FUNCTION_BLOCK FB_FaultHandler
(* 
The faulthandler is responsible for 
	- providing the means for objects to register their faults
	- reporting the active fault types (i.e., message, fatal fault, etc.) --> arActiveFaultTypes
	- providing the means to reset a fault type
	- keeping a log of all faults

It is not responsible for
	- resetting the actual fault (this is up to the object that registered the fault)
	- handling any HMI related functionality

Active faults do not disappear from the log, the need to be manually cleared by issuing a CmdReset and CmdClearInactive.
*)
VAR CONSTANT
	MAX_FAULTS_IN_LOG : UINT := 10;
END_VAR
VAR_INPUT
	nMaxInactiveCycles : UINT := 50; // Once faults haven't been activated for a number of PLC cycles, deactivate them. 0 = do not automatically deactivate faults 
END_VAR
VAR_OUTPUT
	arFaultLog 			: ARRAY [1..MAX_FAULTS_IN_LOG] OF UDT_FaultLogItem;
	nFaultsInLog 		: UINT;
	nActiveFaults 		: UINT;
	arActiveFaultTypes 	: ARRAY[0..(E_FaultTypes._ENUM_SIZE - 1)] OF BOOL; // Status of each fault type
END_VAR
VAR
	bCmdReset : BOOL;
	eResetState : E_ResetState;
	arActiveFaultTypes_Internal : ARRAY[0..(E_FaultTypes._ENUM_SIZE - 1)] OF BOOL; // The actual status of each fault type, which is reported unless the reset cycle is active
	
	nLogIndex : UINT; // Array index of the last added item in the log (zero until the first item arrives)
	nIterIndex : UINT; // Index of the fault log iterator (used for properties First and Next)
END_VAR

UpdateInactiveCycles();

ExecReset();

UpdateActiveFaultStatus();

METHOD PUBLIC CmdAddFault : BOOL
(*
CmdAddFault should be called every cycle.
If the fault is active, it's corresponding fault type is enabled.
Updates the fault log.
*)
VAR_IN_OUT
	stFault : UDT_Fault; // active fault structure input
END_VAR
VAR_INPUT
	stIdentity : UDT_Identity;
END_VAR
// Update the log
UpdateLog(stFault, stIdentity);
END_METHOD

METHOD PUBLIC CmdClearInactive : BOOL // Remove inactive faults from the log
VAR
	stEmptyItem : UDT_FaultLogItem;
	i : UINT; // Iterator
END_VAR
nFaultsInLog := MAX_FAULTS_IN_LOG;
IF (eResetState = E_ResetState.Idle) THEN
	FOR i := 1 TO MAX_FAULTS_IN_LOG DO
		IF (NOT arFaultLog[i].stFault.Active) THEN
			nFaultsInLog :=nFaultsInLog - 1;
			arFaultLog[i] := stEmptyItem;
			arFaultLog[i].bEmpty := TRUE;
		END_IF
	END_FOR
	CmdClearInactive := TRUE;
ELSE
	CmdClearInactive := FALSE;
END_IF
END_METHOD

METHOD PUBLIC CmdReset : BOOL // Reset faults; caller is responsible for stopping the call once TRUE is returned
VAR_INPUT
END_VAR
// Trigger the reset cycle
IF (eResetState = E_ResetState.Idle) THEN
	bCmdReset := TRUE;
END_IF

CmdReset := (eResetState = E_ResetState.Done); // Let the caller know when the reset cycle is finished
END_METHOD

METHOD PRIVATE ExecReset : BOOL
VAR
	i : UINT; // Iterator
END_VAR
CASE eResetState OF
	E_ResetState.Idle: // Wait for reset command
		IF bCmdReset THEN
			// Start the reset cycle
			bCmdReset := FALSE;
			eResetState := E_ResetState.ResetFaultTypes;
		ELSE
			ReportActiveFaultStatus();
		END_IF
	E_ResetState.ResetFaultTypes: 
		// During a reset, the active fault types are not updated 
		// This avoids that faults are not reported for 1 PLC cycle, even though they are still active
		// We do however clear the internal fault types, which are updated automatically during the WaitForFaults state.
		FOR i:= 0 TO (E_FaultTypes._ENUM_SIZE - 1) DO		
			arActiveFaultTypes_Internal[i] := FALSE;
		END_FOR
		eResetState := E_ResetState.WaitForFaults;

	E_ResetState.WaitForFaults: // Allow the PLC one cycle to re-add faults
		eResetState := E_ResetState.Done;

	E_ResetState.Done: // Done, report & allow caller one cycle to reset itself
		ReportActiveFaultStatus();
		eResetState := E_ResetState.Idle;
END_CASE
END_METHOD

METHOD PRIVATE FindNonEmptyFault : UINT // Update nIterIndex to first non-empy fault (if available)
VAR_INPUT
	nStartIndex : UINT;
END_VAR
VAR
	i : UINT; // Iterator
END_VAR
// Sanitize input
nStartIndex := LIMIT(1, nStartIndex, MAX_FAULTS_IN_LOG);

// Iterate array backwards until a non empty item is found.
FOR i := 1 TO MAX_FAULTS_IN_LOG DO
	IF arFaultLog[nStartIndex].bEmpty THEN
		nStartIndex := nStartIndex - 1;
		IF nStartIndex = 0 THEN
			nStartIndex := MAX_FAULTS_IN_LOG;
		END_IF
	ELSE
		EXIT;
	END_IF
END_FOR

FindNonEmptyFault := nStartIndex;
END_METHOD

PROPERTY PUBLIC Head : UDT_FaultLogItem // Returns the head of the log (the latest item added)
GET
nIterIndex := FindNonEmptyFault(nLogIndex);
Head := arFaultLog[nIterIndex];
END_GET
SET
END_SET
END_PROPERTY

PROPERTY PUBLIC Next : UDT_FaultLogItem // Get the next item in the log (travelling backwards through the array)
GET
nIterIndex := FindNonEmptyFault(nIterIndex - 1);
Next := arFaultLog[nIterIndex];
END_GET
SET
END_SET
END_PROPERTY

METHOD PRIVATE ReportActiveFaultStatus : BOOL // Update active fault types based on active faults in the log
VAR
	i : UINT; // Iterator
END_VAR
// Report the status of each fault type to outside world	
FOR i:= 0 TO (E_FaultTypes._ENUM_SIZE - 1) DO		
	arActiveFaultTypes[i] := arActiveFaultTypes_Internal[i];
END_FOR
END_METHOD

METHOD PRIVATE UpdateActiveFaultStatus : BOOL // Update active fault types based on active faults in the log
VAR
	i : UINT; // Iterator
END_VAR
// Get active faults from log
nActiveFaults := 0;
FOR i := 1 TO MAX_FAULTS_IN_LOG DO
	IF (arFaultLog[i].stFault.Active) THEN 
		// Update the number of active faults
		nActiveFaults := nActiveFaults + 1;
		// Update active fault type feedback
		arActiveFaultTypes_Internal[arFaultLog[i].stFault.FaultType] := TRUE; 
	END_IF
END_FOR
END_METHOD

METHOD PRIVATE UpdateInactiveCycles : BOOL // Update the number of inactive cycles, and deactive fault once it reaches the max number of inactive cycles
VAR
	i : UINT; // Iterator
END_VAR
IF (nMaxInactiveCycles > 0) THEN
	FOR i := 1 TO MAX_FAULTS_IN_LOG DO
		IF arFaultLog[i].stFault.Active THEN
			arFaultLog[i].nInactiveCycles := MIN(16#FFFF, arFaultLog[i].nInactiveCycles + 1);
			IF (arFaultLog[i].nInactiveCycles > nMaxInactiveCycles) THEN
				arFaultLog[i].stFault.Active := FALSE;
				arFaultLog[i].EndTime := Sys_Variables.SystemTime;	
			END_IF
		END_IF
	END_FOR
END_IF
END_METHOD

METHOD PRIVATE UpdateLog : BOOL
(*
Update the fault log array. 
If a fault becomes active, it is added to the array and the start time is updated.
If a fault stops being active, the end time is updated.
Inactive faults are cleared by CmdReset.
*)
VAR_IN_OUT
	stFault : UDT_Fault;
END_VAR
VAR_INPUT
	stIdentity : UDT_Identity;
END_VAR
VAR
	sId : STRING;
	nFaultIndexInLog : UINT;
	i : UINT; // Iterator
END_VAR
// Check if the fault already exists in the log. 
// For this, we need to compare the description and the fault ID.

// First, build the fault ID
sId := TO_STRING(stFault.FaultType);
sId := CONCAT(sId,'.');
IF stIdentity.nParentId > 0 THEN
	sId := CONCAT(sId,UDINT_TO_STRING(stIdentity.nParentId));
	sId := CONCAT(sId,'.');
END_IF
sId := CONCAT(sId,UINT_TO_STRING(stIdentity.nId));
sId := CONCAT(sId,'.');
sId := CONCAT(sId,UDINT_TO_STRING(stIdentity.eComponentType));
sId := CONCAT(sId,'.');
sId := CONCAT(sId,stIdentity.sName);

// Now check if the fault already exists in the log
FOR i := 1 TO MAX_FAULTS_IN_LOG DO
	IF (NOT arFaultLog[i].bEmpty) 
		AND (arFaultLog[i].Id = sId) 
		AND (arFaultLog[i].stFault.Description = stFault.Description)
		AND (ANY_TO_DWORD(arFaultLog[i].EndTime) = 0)
	THEN // Found fault in the log
		nFaultIndexInLog := i;
		EXIT; // No need to iterate any further
	END_IF
END_FOR

IF nFaultIndexInLog > 0 THEN // Already exists in the log
	IF (stFault.Active) THEN // Still active, reset inactive cycle counter
		arFaultLog[nFaultIndexInLog].nInactiveCycles := 0;
	ELSIF (ANY_TO_DWORD(arFaultLog[nFaultIndexInLog].EndTime) = 0) THEN // No longer active, update end time and active state
		arFaultLog[nFaultIndexInLog].stFault.Active := FALSE;
		arFaultLog[nFaultIndexInLog].EndTime := Sys_Variables.SystemTime;
	END_IF
ELSIF stFault.Active THEN // New active fault, add it to the log
	// Update the log index (if full, move to beginning of the log)
	nLogIndex := (nLogIndex MOD MAX_FAULTS_IN_LOG) + 1;
	nFaultsInLog := MIN(nFaultsInLog + 1, MAX_FAULTS_IN_LOG);
	// Copy to log and update start time
	arFaultLog[nLogIndex].bEmpty := FALSE;
	arFaultLog[nLogIndex].stFault := stFault;
	arFaultLog[nLogIndex].Id := sId;
	arFaultLog[nLogIndex].StartTime := Sys_Variables.SystemTime;
	arFaultLog[nLogIndex].EndTime := ANY_TO_DT(0);
	arFaultLog[nLogIndex].nInactiveCycles := 0;
END_IF
END_METHOD

END_FUNCTION_BLOCK

(* stored: Version 1.1.0.1, ProductVersion 3.1.4024.11
   POU FB_FaultHandler: Id {08f65884-c647-4a29-b7ba-51d088979c07}, SpecialFunc None
   Folder Private: Id {2e728eb6-79bc-4de8-8875-9d08a8df9edd}
   Method CmdAddFault: Id {cd103280-aca4-4b4a-a070-10b84eec5ffb}
   Method CmdClearInactive: Id {3ab26ba4-92e5-0c92-3fbe-58c7f26971b2}
   Method CmdReset: Id {a9c5d6bc-61dd-41fc-99d9-5b14d5fa2712}
   Method ExecReset: Id {5409ab96-3bb3-0061-05e8-ad57d1261a31}
   Method FindNonEmptyFault: Id {f653cfda-c6a2-0aba-0999-a219be313e66}
   Property Head: Id {51df95bf-2d5c-0e2f-1669-066486ace38d}
   Get Get: Id {5da39590-30a9-04b4-307b-1dd3ceac2537}
   Set Set: Id {f26a9a04-102d-0fab-2b21-bb756981a144}
   Property Next: Id {3bc770ea-8ea7-000b-0986-7649ccc14e3e}
   Get Get: Id {fcd54202-6b03-0138-1a15-35466f1589c9}
   Set Set: Id {cac173bd-6bf0-0aee-34ab-d083a619fe0b}
   Method ReportActiveFaultStatus: Id {bb238a89-dedc-03ce-36d6-86f48f05fe0e}
   Method UpdateActiveFaultStatus: Id {478e9522-b643-0b3d-0d6d-947b92d13a5f}
   Method UpdateInactiveCycles: Id {e86406ea-3c11-02d6-1216-7a9b59f97c40}
   Method UpdateLog: Id {9b29b2d1-5975-05b2-2182-eff98e668948} *)
